// TIA Portal V20 export
TYPE "BarrerasGating"
   STRUCT
      DesActivar : Bool;
      EnTension : Bool;
      S_Rearme : Bool;
      S_TestLuces : Bool;
      InicioGating : Bool;
      FinalGating : Bool;
      Retardo_InicioGating : Time := T#200ms;
      Retardo_FinalGating : Time := T#200ms;
      V_MaximoGating : Time := T#30s;
   END_STRUCT;
END_TYPE
